{attribute addProperty BoxType "EL5072-0000-0016"}
{attribute addProperty Id "IND_Inputs_ChannelAT %I*ARRAY[0..3] OF IND_Inputs_Channel_F11037BF160200IND_Outputs_ChannelAT %Q*ARRAY[0..4] OF IND_Outputs_Channel_CDB9543D112140WcStateAT %I*WcState_98A4DF7520.250InfoDataAT %I*InfoData_BC63D37F80100"}
{attribute addProperty CRC "329872429"}
{attribute addProperty SizeInBites "354"}
{attribute addProperty SizeInBytes "44.25"}
TYPE EL5072_762C412B :
STRUCT
	{attribute addProperty Name "IND_Inputs_Channel"}
	IND_Inputs_Channel : ARRAY[0..3] OF IND_Inputs_Channel_F11037BF;
	{attribute addProperty Name "IND_Outputs_Channel"}
	IND_Outputs_Channel : ARRAY[0..4] OF IND_Outputs_Channel_CDB9543D;
	{attribute addProperty Name "WcState"}
	WcState : WcState_98A4DF75;
	{attribute addProperty Name "InfoData"}
	InfoData : InfoData_BC63D37F;
END_STRUCT
END_TYPE

(* stored: Version 1.2.0.0, ProductVersion 3.1.4024.9
   DUT EL5072_762C412B: Id {83f3d787-13fe-41b2-8e2b-e4b5327a3618} *)
